// SIMATIC S7-200 project (STEP 7-Micro/WIN), CPU 224 REL 02.01

ORGANIZATION_BLOCK MAIN:OB1
TITLE=PROGRAM COMMENTS
BEGIN
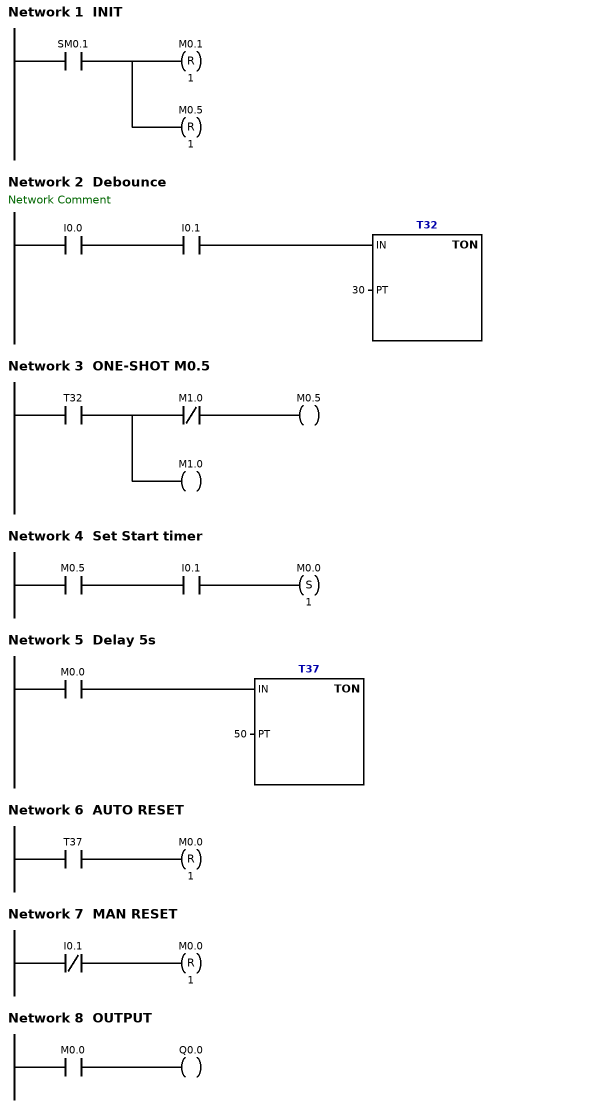
Network 1 // INIT
LD     SM0.1
R      M0.1, 1
R      M0.5, 1
Network 2 // Debounce
// Network Comment
LD     I0.0
A      I0.1
TON    T32, 30
Network 3 // ONE-SHOT M0.5
LD     T32
LPS
AN     M1.0
=      M0.5
LPP
=      M1.0
Network 4 // Set Start timer
LD     M0.5
A      I0.1
S      M0.0, 1
Network 5 // Delay 5s
LD     M0.0
TON    T37, 50
Network 6 // AUTO RESET
LD     T37
R      M0.0, 1
Network 7 // MAN RESET
LDN    I0.1
R      M0.0, 1
Network 8 // OUTPUT
LD     M0.0
=      Q0.0
END_ORGANIZATION_BLOCK
